	//==============================================================
	// EN: Stack buffer conveyor control
	// PT: Controle das esteiras buffer de pilhas
	//==============================================================
	stackBufferControlState                 : INT;
	stackBufferTargetConveyor               : INT;
	elevatorStackExitClearSensorOld         : BOOL;
	rElevatorStackExitClear                 : BOOL;
	tonStackBufferStopDelay                 : TON;
	tonStackBufferTransferTimeout           : TON;
	tonStackBufferFullSpeedReduction        : TON;
	stackBufferTransferTimeoutPulse         : BOOL;
	
	instTONPaperPressOff: TON;
	instTONPaperPressOn: TON;
	paperPressOnPhase: BOOL;

	// EN: Delays exhaust fan shutdown after line speed drops.
	// PT: Atrasa o desligamento do exaustor após a queda da velocidade da linha.
	instTONSheetConveyor1ExhaustFanStopDelay : TON;
END_VAR

_SystemControl();

_SheetConveyorGroupControl();
_ConveyorSpeedControl();
_SheetConveyor1ExhaustFanControl();

_SheetStackDischargeControl();

_BackstopControl();
_ElevatorControl();
_SheetStackAlignmentBrushControl();
_SheetStackDischargeConveyorControl();
_StackBufferConveyorsControl();
_SheetBrushControl();
_paperPressControl();
_MachineAuxiliary();
_HmiStatus();
_AlarmControl();

//==============================================================
// COMPLEX STACKER — ALARM CONTROL
// EN: Maps internal faults and status conditions to HMI alarm structure.
//==============================================================
METHOD _AlarmControl

VAR
	alarmCompareResult                         : DINT;
	elevatorHomeReleasePermissivesWithoutBackstop : BOOL;
	elevatorUpBlockedByBackstopCondition       : BOOL;
	elevatorUpPermissivesWithoutBackstop       : BOOL;
	elevatorUpRequestActive                    : BOOL;
	hmiAlarmsNotActive                         : hmiAlarmsComplexStacker_TypeStruct;
END_VAR
//==============================================================
// HMI alarms reset / latch logic
//==============================================================

// EN: Detect an actual upward request before the backstop material sensor
//     is applied to the elevator movement permissive.
// PT: Detecta um pedido real de subida antes de aplicar o sensor de material
//     do backstop ao permissivo de movimento do elevador.
elevatorUpRequestActive :=
    (
        (elevatorControlState = 11) AND
        elevatorHomeLimitReached
    ) OR
    (
        (elevatorControlState = 14) AND
        elevatorHomeDischargeComplete AND
        NOT elevatorInPosition AND
        (elevatorRawSpeedRefMmps > 0.0)
    ) OR
    (
        (elevatorControlState = 20) AND
        elevatorManualCommandRequest AND
        elevatorUpCmd AND
        NOT elevatorDownCmd
    ) OR
    (
        (elevatorControlState = 40) AND
        elevatorTargetOverrideActive AND
        NOT elevatorInPosition AND
        (elevatorRawSpeedRefMmps > 0.0)
    );


elevatorUpPermissivesWithoutBackstop :=
    systemRunEnable AND
    safetyCircuitOk AND
    elevatorDriveOk AND
    NOT elevatorFault AND
    NOT elevatorUpperLimit AND
    NOT elevatorUpperSafetyLimit AND
    (
        NOT elevatorHomed OR
        (elevatorPositionMm < machineConfig.elevatorMaxPositionMm)
    );


elevatorHomeReleasePermissivesWithoutBackstop :=
    systemRunEnable AND
    safetyCircuitOk AND
    elevatorDriveOk AND
    NOT elevatorFault AND
    NOT elevatorUpperLimit AND
    NOT elevatorUpperSafetyLimit;


elevatorUpBlockedByBackstopCondition :=
    backstopMaterialInterlockSensor AND
    (
        (
            (elevatorControlState = 11) AND
            elevatorHomeLimitReached AND
            elevatorHomeReleasePermissivesWithoutBackstop
        ) OR
        (
            (elevatorControlState <> 11) AND
            elevatorUpRequestActive AND
            elevatorUpPermissivesWithoutBackstop
        )
    );


// EN: A short delay avoids latching the alarm because of sensor bounce.
// PT: Um pequeno atraso evita memorizar o alarme devido a repique do sensor.
tonElevatorUpBlockedByBackstopAlarm(
    IN := elevatorUpBlockedByBackstopCondition,
    PT := T#500MS
);

IF resetCmd THEN

    // Reset geral dos alarmes
    hmiAlarms := hmiAlarmsNotActive;

ELSE

    //==============================================================
    // 1) General / system alarms
    //==============================================================
    hmiAlarms.safetyCircuitNotOk :=
        hmiAlarms.safetyCircuitNotOk OR
        NOT safetyCircuitOk;

    hmiAlarms.systemFaultActive :=
        hmiAlarms.systemFaultActive OR
        faultActive OR
        (
            backstopRequiredForAutomaticOperation AND
            backstopFault
        ) OR
        elevatorFault OR
        sheetStackDischargeFault OR
        sheetStackDischargeConveyorFault OR
        NOT stackBufferConveyor1DriveOk OR
        NOT stackBufferConveyor2DriveOk OR
        NOT stackBufferConveyor3DriveOk OR
        stackBufferTransferTimeoutPulse;

    hmiAlarms.systemNotEnabled :=
        hmiAlarms.systemNotEnabled OR
        NOT systemRunEnable;

    // EN: These generic safety feedbacks are used only for diagnostics.
    // PT: Estes retornos genéricos de segurança são usados apenas para diagnóstico.
    hmiAlarms.safetyFeedback1NotOk := hmiAlarms.safetyFeedback1NotOk OR NOT safetyFeedBack1;
    hmiAlarms.safetyFeedback2NotOk := hmiAlarms.safetyFeedback2NotOk OR NOT safetyFeedBack2;
    hmiAlarms.safetyFeedback3NotOk := hmiAlarms.safetyFeedback3NotOk OR NOT safetyFeedBack3;
    hmiAlarms.safetyFeedback4NotOk := hmiAlarms.safetyFeedback4NotOk OR NOT safetyFeedBack4;
    hmiAlarms.safetyFeedback5NotOk := hmiAlarms.safetyFeedback5NotOk OR NOT safetyFeedBack5;
    hmiAlarms.safetyFeedback6NotOk := hmiAlarms.safetyFeedback6NotOk OR NOT safetyFeedBack6;
    hmiAlarms.safetyFeedback7NotOk := hmiAlarms.safetyFeedback7NotOk OR NOT safetyFeedBack7;
    hmiAlarms.safetyFeedback8NotOk := hmiAlarms.safetyFeedback8NotOk OR NOT safetyFeedBack8;


    //==============================================================
    // 2) Sheet conveyor group alarms
    //==============================================================
    hmiAlarms.sheetConveyor1DriveNotOk :=
        hmiAlarms.sheetConveyor1DriveNotOk OR
        NOT sheetConveyor1DriveOk;

    hmiAlarms.sheetConveyor2DriveNotOk :=
        hmiAlarms.sheetConveyor2DriveNotOk OR
        NOT sheetConveyor2DriveOk;

    hmiAlarms.sheetConveyor3DriveNotOk :=
        hmiAlarms.sheetConveyor3DriveNotOk OR
        NOT sheetConveyor3DriveOk;

    hmiAlarms.sheetConveyor4DriveNotOk :=
        hmiAlarms.sheetConveyor4DriveNotOk OR
        NOT sheetConveyor4DriveOk;

    hmiAlarms.sheetConveyorGroupFault :=
        hmiAlarms.sheetConveyorGroupFault OR
        NOT safetyCircuitOk OR
        NOT sheetConveyor1DriveOk OR
        NOT sheetConveyor2DriveOk OR
        NOT sheetConveyor3DriveOk OR
        NOT sheetConveyor4DriveOk;


    //==============================================================
    // 2.1) Stack buffer conveyor alarms
    // EN: Buffer drive faults are alarmed without stopping the main
    //     synchronized conveyor group automatically.
    // PT: Falhas dos drives do buffer geram alarme sem parar automaticamente
    //     o grupo principal de esteiras sincronizadas.
    //==============================================================
    hmiAlarms.stackBufferConveyor1DriveNotOk :=
        hmiAlarms.stackBufferConveyor1DriveNotOk OR
        NOT stackBufferConveyor1DriveOk;

    hmiAlarms.stackBufferConveyor2DriveNotOk :=
        hmiAlarms.stackBufferConveyor2DriveNotOk OR
        NOT stackBufferConveyor2DriveOk;

    hmiAlarms.stackBufferConveyor3DriveNotOk :=
        hmiAlarms.stackBufferConveyor3DriveNotOk OR
        NOT stackBufferConveyor3DriveOk;

    hmiAlarms.stackBufferConveyorGroupFault :=
        hmiAlarms.stackBufferConveyorGroupFault OR
        NOT safetyCircuitOk OR
        NOT stackBufferConveyor1DriveOk OR
        NOT stackBufferConveyor2DriveOk OR
        NOT stackBufferConveyor3DriveOk;

    hmiAlarms.stackBufferTransferTimeout :=
        hmiAlarms.stackBufferTransferTimeout OR
        stackBufferTransferTimeoutPulse;

    hmiAlarms.stackBufferFull :=
        hmiAlarms.stackBufferFull OR
        stackBufferFull;

    hmiAlarms.stackBufferSpeedReductionActive :=
        hmiAlarms.stackBufferSpeedReductionActive OR
        lineSpeedReductionRequest;

 //   hmiAlarms.synchronizedConveyorsNotRunning :=
 //       hmiAlarms.synchronizedConveyorsNotRunning OR
 //       (
 //           systemRunEnable AND
 //           NOT synchronizedConveyorsRunning
 //       );


    //==============================================================
    // 3) Sheet stack separation alarms / indications
    //==============================================================
    // Mantido comentado conforme lógica original.
    // Se quiser ativar como latch, use o mesmo padrão:
    //
    // hmiAlarms.sheetStackSeparationNotReady :=
    //     hmiAlarms.sheetStackSeparationNotReady OR
    //     (
    //         systemRunEnable AND
    //         synchronizedConveyorsRunning AND
    //         NOT sheetStackSeparationReady
    //     );
    //
    // hmiAlarms.sheetStackSeparationActive :=
    //     hmiAlarms.sheetStackSeparationActive OR
    //     sheetStackSeparationActive;
    //
    // hmiAlarms.sheetStackBrakeActive :=
    //     hmiAlarms.sheetStackBrakeActive OR
    //     sheetStackBrakeActive;


    //==============================================================
    // 4) Sheet stack discharge sequence alarms / indications
    //==============================================================
    hmiAlarms.sheetStackDischargeFault :=
        hmiAlarms.sheetStackDischargeFault OR
        sheetStackDischargeFault;

    hmiAlarms.sheetStackDischargeLastCycleNotOk :=
        hmiAlarms.sheetStackDischargeLastCycleNotOk OR
        (
            NOT sheetStackDischargeLastCycleOk AND
            sheetStackDischargeLastResultCode <> 0
        );

    hmiAlarms.sheetStackDischargeTimeout :=
        hmiAlarms.sheetStackDischargeTimeout OR
        (
            sheetStackDischargeFault AND
            (sheetStackDischargeLastResultCode = 3)
        );

    hmiAlarms.sheetStackDischargeManualSkip :=
        hmiAlarms.sheetStackDischargeManualSkip OR
        sheetStackDischargeLastResultCode = 2;

    hmiAlarms.sheetStackDischargeWaitSeparationTimeout :=
        hmiAlarms.sheetStackDischargeWaitSeparationTimeout OR
        (
            sheetStackDischargeFault AND
            (sheetStackDischargeLastFaultCode = 10)
        );

    hmiAlarms.sheetStackDischargePositioningTimeout :=
        hmiAlarms.sheetStackDischargePositioningTimeout OR
        (
            sheetStackDischargeFault AND
            (sheetStackDischargeLastFaultCode = 20)
        );

    hmiAlarms.sheetStackDischargeConveyorStartTimeout :=
        hmiAlarms.sheetStackDischargeConveyorStartTimeout OR
        (
            sheetStackDischargeFault AND
            (sheetStackDischargeLastFaultCode = 30)
        );

    hmiAlarms.sheetStackDischargePlatformClearTimeout :=
        hmiAlarms.sheetStackDischargePlatformClearTimeout OR
        (
            sheetStackDischargeFault AND
            (sheetStackDischargeLastFaultCode = 31)
        );

    hmiAlarms.sheetStackDischargeReturnTimeout :=
        hmiAlarms.sheetStackDischargeReturnTimeout OR
        (
            sheetStackDischargeFault AND
            (sheetStackDischargeLastFaultCode = 50)
        );


    //==============================================================
    // 5) Sheet stack discharge conveyor alarms
    //==============================================================
    hmiAlarms.sheetStackDischargeConveyorDriveNotOk :=
        hmiAlarms.sheetStackDischargeConveyorDriveNotOk OR
        NOT sheetStackDischargeConveyorDriveOk;

    hmiAlarms.sheetStackDischargeConveyorFault :=
        hmiAlarms.sheetStackDischargeConveyorFault OR
        sheetStackDischargeConveyorFault;


    //==============================================================
    // 6) Backstop alarms / indications
    //==============================================================
    hmiAlarms.backstopDriveNotOk :=
        hmiAlarms.backstopDriveNotOk OR
        NOT backstopDriveOk;

    hmiAlarms.backstopFault :=
        hmiAlarms.backstopFault OR
        backstopFault;

    hmiAlarms.backstopNotHomed :=
        hmiAlarms.backstopNotHomed OR
        (
            systemRunEnable AND
            backstopAutoCmd AND
            NOT backstopHomed AND
            NOT backstopAutoHomePending AND
            NOT (
                (backstopControlState >= 10) AND
                (backstopControlState <= 14)
            )
        );

    hmiAlarms.backstopHomingTimeout :=
        hmiAlarms.backstopHomingTimeout OR
        (
            backstopFault AND
            (backstopFaultCode = 3)
        );

    hmiAlarms.backstopInvalidHomeDirection :=
        hmiAlarms.backstopInvalidHomeDirection OR
        (
            backstopFault AND
            (backstopFaultCode = 5)
        );

    (*
    hmiAlarms.backstopNotInPosition :=
        hmiAlarms.backstopNotInPosition OR
        (
            systemRunEnable AND
            backstopAutoCmd AND
            backstopHomed AND
            NOT backstopInPosition AND
            NOT backstopTargetOverrideActive
        );
    *)

    hmiAlarms.backstopSafeMaxLimitActive :=
        hmiAlarms.backstopSafeMaxLimitActive OR
        backstopSafeMaxLimit;

    hmiAlarms.backstopSafeMinLimitActive :=
        hmiAlarms.backstopSafeMinLimitActive OR
        backstopSafeMinLimit;

    (*
    hmiAlarms.backstopMaxLimitActive :=
        hmiAlarms.backstopMaxLimitActive OR
        backstopMaxLimit;

    hmiAlarms.backstopMinLimitActive :=
        hmiAlarms.backstopMinLimitActive OR
        backstopMinLimit;

    hmiAlarms.backstopManualInterventionActive :=
        hmiAlarms.backstopManualInterventionActive OR
        backstopManualInterventionActive;
    *)


    //==============================================================
    // 7) Elevator alarms / indications
    //==============================================================
    hmiAlarms.elevatorDriveNotOk :=
        hmiAlarms.elevatorDriveNotOk OR
        NOT elevatorDriveOk;

    hmiAlarms.elevatorFault :=
        hmiAlarms.elevatorFault OR
        elevatorFault;

    hmiAlarms.elevatorNotHomed :=
        hmiAlarms.elevatorNotHomed OR
        (
            systemRunEnable AND
            elevatorAutoCmd AND
            NOT elevatorHomed AND
            NOT elevatorAutoHomePending AND
            NOT (
                (elevatorControlState >= 10) AND
                (elevatorControlState <= 14)
            )
        );

    hmiAlarms.elevatorHomingTimeout :=
        hmiAlarms.elevatorHomingTimeout OR
        (
            elevatorFault AND
            (elevatorFaultCode = 3)
        );

    hmiAlarms.elevatorUpBlockedByBackstopMaterialInterlock :=
        hmiAlarms.elevatorUpBlockedByBackstopMaterialInterlock OR
        tonElevatorUpBlockedByBackstopAlarm.Q;

//    hmiAlarms.elevatorNotInPosition :=
//        hmiAlarms.elevatorNotInPosition OR
//        (
//            systemRunEnable AND
//            elevatorAutoCmd AND
//            elevatorHomed AND
//            NOT elevatorInPosition
//        );

    hmiAlarms.elevatorUpperSafetyLimitActive :=
        hmiAlarms.elevatorUpperSafetyLimitActive OR
        elevatorUpperSafetyLimit;

    hmiAlarms.elevatorLowerSafetyLimitActive :=
        hmiAlarms.elevatorLowerSafetyLimitActive OR
        elevatorLowerSafetyLimit;

    (*
    hmiAlarms.elevatorUpperLimitActive :=
        hmiAlarms.elevatorUpperLimitActive OR
        elevatorUpperLimit;

    hmiAlarms.elevatorLowerLimitActive :=
        hmiAlarms.elevatorLowerLimitActive OR
        elevatorLowerLimit;
    *)

END_IF;


// EN: The general output follows every latched field in the alarm structure.
// PT: A saída geral acompanha qualquer campo memorizado na estrutura de alarmes.
alarmCompareResult := MEMCMP(
    pBuf1 := ADR(hmiAlarmsNotActive),
    pBuf2 := ADR(hmiAlarms),
    n := SIZEOF(hmiAlarms)
);

alarmActive := alarmCompareResult <> 0;
END_METHOD

//==============================================================
// COMPLEX STACKER — BACKSTOP CONTROL
// EN: Controls the backstop axis with homing, manual movement,
//     automatic positioning, override positioning and protections.
//
// Signed speed convention:
// Positive = open
// Negative = close
//
// State code:
// 0  = STOP
// 10 = HOME_FAST_SEARCH
// 11 = HOME_SLOW_EXIT_SENSOR
// 12 = HOME_SET_ENCODER
// 13 = HOME_WAIT_AFTER_SET
// 14 = HOME_MOVE_TO_TARGET
// 20 = MANUAL
// 30 = AUTO_POSITION
// 40 = FAULT
//==============================================================
METHOD _BackstopControl



//==============================================================
// 1) Default internal commands
//==============================================================
// EN: Internal signed speed is reset every scan and set by the active state.
//     Positive = open, negative = close.
backstopSignedSpeedRefMmps := 0.0;

// EN: Internal trigger for encoder set pulse.
backstopSetEncoderPositionTrigger := FALSE;


//==============================================================
// 2) Edge detection
//==============================================================
// EN: Home can be requested manually by HMI or automatically by _SystemControl.
//     Automatic home is accepted only when backstopAutoCmd is enabled.
//     Movement is allowed only when master system run is enabled.
backstopHomeRequestCombined :=
    systemRunEnable AND
    (
        backstopHomeCmd OR
        (
            backstopAutoCmd AND
            backstopAutoHomeRequest
        )
    );

// EN: The automatic pulse is accepted directly so a maintained manual home
//     command cannot hide the mandatory start-triggered request.
// PT: O pulso automático é aceito diretamente para que um comando manual de
//     home mantido não esconda o pedido obrigatório gerado pela partida.
rBackstopHome :=
    (
        backstopHomeRequestCombined AND
        NOT backstopHomeRequestCombinedOld
    ) OR
    (
        systemRunEnable AND
        backstopAutoCmd AND
        backstopAutoHomeRequest
    );

backstopHomeRequestCombinedOld :=
    backstopHomeRequestCombined;


// EN: Execute positioning command edge.
//     This command only generates movement when system is enabled and backstop auto is enabled.
rBackstopExecutePositioning :=
    systemRunEnable AND
    backstopExecutePositioningCmd AND
    NOT backstopExecutePositioningCmdOld;

backstopExecutePositioningCmdOld := backstopExecutePositioningCmd;


// EN: Override falling edge.
//     Used as fallback to return to programmed position if override is released.
backstopTargetOverrideFallingEdge :=
    backstopTargetOverrideOld AND NOT backstopTargetOverrideActive;

backstopTargetOverrideOld := backstopTargetOverrideActive;


//==============================================================
// 3) Home limit selection and edge detection
//==============================================================
// EN: Home limit depends on configured homing direction.
IF machineConfig.backstopHomeDirection > 0 THEN

    backstopHomeLimitReached := backstopMaxLimit;

ELSIF machineConfig.backstopHomeDirection < 0 THEN

    backstopHomeLimitReached := backstopMinLimit;

ELSE

    backstopHomeLimitReached := FALSE;

END_IF;


// EN: Falling edge is used after the home limit has been reached.
backstopHomeLimitFallingEdge :=
    backstopHomeLimitOld AND NOT backstopHomeLimitReached;

backstopHomeLimitOld := backstopHomeLimitReached;


//==============================================================
// 4) Movement permissions
//==============================================================
backstopOpenAllowed :=
    systemRunEnable AND
    safetyCircuitOk AND
    backstopDriveOk AND
    NOT backstopMaxLimit AND
    NOT backstopSafeMaxLimit AND
    (
        (NOT backstopHomed) OR
        (backstopPositionMm < machineConfig.backstopMaxPositionMm)
    );

backstopCloseAllowed :=
    systemRunEnable AND
    safetyCircuitOk AND
    backstopDriveOk AND
    NOT backstopMinLimit AND
    NOT backstopSafeMinLimit AND
    (
        (NOT backstopHomed) OR
        (backstopPositionMm > machineConfig.backstopMinPositionMm)
    );


// EN: During homing, the normal home limit is allowed.
//     Only the safe limit blocks movement.
IF machineConfig.backstopHomeDirection > 0 THEN

    backstopHomeMoveAllowed :=
        systemRunEnable AND
        safetyCircuitOk AND
        backstopDriveOk AND
        NOT backstopSafeMaxLimit;

ELSIF machineConfig.backstopHomeDirection < 0 THEN

    backstopHomeMoveAllowed :=
        systemRunEnable AND
        safetyCircuitOk AND
        backstopDriveOk AND
        NOT backstopSafeMinLimit;

ELSE

    backstopHomeMoveAllowed := FALSE;

END_IF;


//==============================================================
// 5) Programmed / override target calculation
//==============================================================
// EN: Programmed target follows sheet length plus mechanical offset.
//     This value can change, but it does not move the backstop by itself.
backstopProgrammedTargetPositionMm :=
    LIMIT(
        machineConfig.backstopMinPositionMm,
        MAX(0.0, sheetLengthMm) + machineConfig.backstopSheetLengthOffsetMm,
        machineConfig.backstopMaxPositionMm
    );


// EN: Before homing, keep the latched target updated with programmed target.
//     This avoids an invalid old target after power-up.
IF NOT backstopHomed THEN

    backstopLatchedTargetPositionMm := backstopProgrammedTargetPositionMm;

END_IF;


//==============================================================
// 5.1) Automatic positioning request handling
//==============================================================
// EN: Auto mode only enables positioning. It does not execute positioning.
//     Normal positioning must be requested by backstopExecutePositioningCmd.
//     Override positioning is requested by the automatic cycle.
IF NOT systemRunEnable THEN

    backstopPositioningRequestActive := FALSE;


ELSIF NOT backstopAutoCmd THEN

    backstopPositioningRequestActive := FALSE;


ELSIF backstopTargetOverrideActive THEN

    // EN: Override has priority. Clear normal positioning request.
    backstopPositioningRequestActive := FALSE;


ELSIF rBackstopExecutePositioning THEN

    // EN: Latch current programmed target only when execute command is received.
    backstopLatchedTargetPositionMm := backstopProgrammedTargetPositionMm;
    backstopPositioningRequestActive := TRUE;


ELSIF backstopTargetOverrideFallingEdge THEN

    // EN: Fallback after override release.
    //     The discharge sequence should normally keep override active
    //     during return. If override is released unexpectedly, return to
    //     programmed position automatically.
    backstopLatchedTargetPositionMm := backstopProgrammedTargetPositionMm;
    backstopPositioningRequestActive := TRUE;

END_IF;


//==============================================================
// 5.2) Active target selection
//==============================================================
// EN: Discharge override is accepted only while the backstop is in automatic.
//     In manual mode the backstop is completely independent from the cycle.
// PT: O override de descarte é aceito somente com o backstop em automático.
//     No modo manual o backstop fica completamente independente do ciclo.
IF systemRunEnable AND
   backstopAutoCmd AND
   backstopTargetOverrideActive THEN

    backstopTargetPositionMm :=
        LIMIT(
            machineConfig.backstopMinPositionMm,
            backstopTargetOverridePositionMm,
            machineConfig.backstopMaxPositionMm
        );

ELSE

    backstopTargetPositionMm :=
        LIMIT(
            machineConfig.backstopMinPositionMm,
            backstopLatchedTargetPositionMm,
            machineConfig.backstopMaxPositionMm
        );

END_IF;


//==============================================================
// 5.4) Home running flag
//==============================================================
IF (backstopControlState = 10) OR
   (backstopControlState = 11) OR
   (backstopControlState = 12) OR
   (backstopControlState = 13) OR
   (backstopControlState = 14) THEN

    backstopHomeRunning := TRUE;

ELSE

    backstopHomeRunning := FALSE;

END_IF;


//==============================================================
// 6) Position error calculation
//==============================================================
backstopPositionErrorMm :=
    backstopTargetPositionMm - backstopPositionMm;

backstopAbsPositionErrorMm :=
    ABS(backstopPositionErrorMm);

backstopInPosition :=
    backstopHomed AND
    (backstopAbsPositionErrorMm <= machineConfig.backstopPositionToleranceMm);


//==============================================================
// 7) Reset fault command
//==============================================================
IF resetCmd THEN

    IF safetyCircuitOk AND
       backstopDriveOk AND
       NOT backstopSafeMaxLimit AND
       NOT backstopSafeMinLimit THEN

        backstopFault := FALSE;
        backstopFaultCode := 0;

        IF backstopControlState = 40 THEN
            backstopControlState := 0;
        END_IF

    END_IF

END_IF;


//==============================================================
// 8) General protection
//==============================================================
IF NOT safetyCircuitOk THEN

    backstopState := 'SAFETY_OFF';

    tonBackstopHomingTimeout(IN := FALSE);
    tonBackstopHomeSettleDelay(IN := FALSE);

    backstopFault := TRUE;
    backstopFaultCode := 2;
    backstopControlState := 40;


ELSIF NOT backstopDriveOk THEN

    backstopState := 'DRIVE_NOT_OK';

    tonBackstopHomingTimeout(IN := FALSE);
    tonBackstopHomeSettleDelay(IN := FALSE);

    backstopFault := TRUE;
    backstopFaultCode := 1;
    backstopControlState := 40;


ELSIF backstopSafeMaxLimit THEN

    backstopState := 'SAFE_MAX_LIMIT';

    tonBackstopHomingTimeout(IN := FALSE);
    tonBackstopHomeSettleDelay(IN := FALSE);

    backstopFault := TRUE;
    backstopFaultCode := 6;
    backstopControlState := 40;


ELSIF backstopSafeMinLimit THEN

    backstopState := 'SAFE_MIN_LIMIT';

    tonBackstopHomingTimeout(IN := FALSE);
    tonBackstopHomeSettleDelay(IN := FALSE);

    backstopFault := TRUE;
    backstopFaultCode := 7;
    backstopControlState := 40;


ELSIF machineConfig.backstopHomeDirection = 0 THEN

    backstopState := 'INVALID_HOME_DIR';

    tonBackstopHomingTimeout(IN := FALSE);
    tonBackstopHomeSettleDelay(IN := FALSE);

    backstopFault := TRUE;
    backstopFaultCode := 5;
    backstopControlState := 40;


ELSIF NOT systemRunEnable THEN

    // EN: Master stop disables movement without generating an axis fault.
    backstopState := 'SYSTEM_DISABLED';

    backstopSignedSpeedRefMmps := 0.0;

    tonBackstopHomingTimeout(IN := FALSE);
    tonBackstopHomeSettleDelay(IN := FALSE);

    backstopPositioningRequestActive := FALSE;

    IF backstopControlState <> 40 THEN
        backstopControlState := 0;
    END_IF


ELSE

    //==============================================================
    // 9) Mode selection
    //==============================================================
    // EN: Homing has priority over manual and automatic positioning.
    IF rBackstopHome AND NOT backstopFault THEN
        backstopControlState := 10;

        // EN: Consume the pending request only after homing is accepted.
        // PT: Consome o pedido pendente somente após o homing ser aceito.
        backstopAutoHomePending := FALSE;
    END_IF;


    //==============================================================
    // 10) Backstop state machine
    //==============================================================
    CASE backstopControlState OF

        0: // STOP
            backstopState := 'STOP';

            tonBackstopHomingTimeout(IN := FALSE);
            tonBackstopHomeSettleDelay(IN := FALSE);

            // EN: Manual is allowed even with auto enabled,
            //     but not during an automatic cycle override.
            IF (backstopOpenCmd OR backstopCloseCmd) AND
               NOT (
                   backstopAutoCmd AND
                   backstopTargetOverrideActive
               ) THEN

                backstopControlState := 20;


            ELSIF backstopAutoCmd AND
                  (
                      backstopTargetOverrideActive OR
                      backstopPositioningRequestActive
                  ) THEN

                backstopControlState := 30;

            END_IF


        10: // HOME_FAST_SEARCH
            backstopState := 'HOME_FAST';

            backstopHomed := FALSE;
            backstopInPosition := FALSE;

            tonBackstopHomeSettleDelay(IN := FALSE);

            tonBackstopHomingTimeout(
                IN := TRUE,
                PT := machineConfig.backstopHomingTimeout
            );

            IF tonBackstopHomingTimeout.Q THEN

                backstopSignedSpeedRefMmps := 0.0;

                tonBackstopHomingTimeout(IN := FALSE);

                backstopFault := TRUE;
                backstopFaultCode := 3;

                backstopState := 'HOME_TIMEOUT';
                backstopControlState := 40;


            ELSIF backstopHomeLimitReached THEN

                backstopSignedSpeedRefMmps := 0.0;

                backstopControlState := 11;


            ELSE

                IF backstopHomeMoveAllowed THEN

                    IF machineConfig.backstopHomeDirection > 0 THEN

                        backstopSignedSpeedRefMmps :=
                            ABS(machineConfig.backstopHomingSpeedMmps);

                    ELSE

                        backstopSignedSpeedRefMmps :=
                            -ABS(machineConfig.backstopHomingSpeedMmps);

                    END_IF

                ELSE

                    backstopSignedSpeedRefMmps := 0.0;

                END_IF

            END_IF


        11: // HOME_SLOW_EXIT_SENSOR
            backstopState := 'HOME_SLOW_EXIT';

            tonBackstopHomeSettleDelay(IN := FALSE);

            tonBackstopHomingTimeout(
                IN := TRUE,
                PT := machineConfig.backstopHomingTimeout
            );

            IF tonBackstopHomingTimeout.Q THEN

                backstopSignedSpeedRefMmps := 0.0;

                tonBackstopHomingTimeout(IN := FALSE);

                backstopFault := TRUE;
                backstopFaultCode := 3;

                backstopState := 'HOME_TIMEOUT';
                backstopControlState := 40;


            ELSIF backstopHomeLimitFallingEdge THEN

                backstopSignedSpeedRefMmps := 0.0;

                tonBackstopHomingTimeout(IN := FALSE);

                backstopControlState := 12;


            ELSE

                IF backstopHomeMoveAllowed THEN

                    IF machineConfig.backstopHomeDirection > 0 THEN

                        backstopSignedSpeedRefMmps :=
                            -ABS(machineConfig.backstopMinMoveSpeedMmps);

                    ELSE

                        backstopSignedSpeedRefMmps :=
                            ABS(machineConfig.backstopMinMoveSpeedMmps);

                    END_IF

                ELSE

                    backstopSignedSpeedRefMmps := 0.0;

                END_IF

            END_IF


        12: // HOME_SET_ENCODER
            backstopState := 'HOME_SET_ENCODER';

            backstopSignedSpeedRefMmps := 0.0;

            tonBackstopHomingTimeout(IN := FALSE);
            tonBackstopHomeSettleDelay(IN := FALSE);

            // EN: Set encoder to configured known home position.
            backstopSetEncoderPositionTrigger := TRUE;
            backstopSetEncoderPositionMm := machineConfig.backstopHomePositionMm;

            backstopHomed := TRUE;
            backstopFault := FALSE;
            backstopFaultCode := 0;

            // EN: After homing, latch current programmed target for home move.
            backstopLatchedTargetPositionMm := backstopProgrammedTargetPositionMm;
            backstopPositioningRequestActive := TRUE;

            // EN: Homing cancels previous manual intervention memory.
            backstopManualInterventionActive := FALSE;
            backstopManualInterventionPositionMm := 0.0;

            backstopControlState := 13;


        13: // HOME_WAIT_AFTER_SET
            backstopState := 'HOME_WAIT';

            backstopSignedSpeedRefMmps := 0.0;

            tonBackstopHomingTimeout(IN := FALSE);

            // EN: Fixed wait after encoder set.
            tonBackstopHomeSettleDelay(
                IN := TRUE,
                PT := T#5S
            );

            IF tonBackstopHomeSettleDelay.Q THEN

                tonBackstopHomeSettleDelay(IN := FALSE);

                backstopControlState := 14;

            END_IF


        14: // HOME_MOVE_TO_TARGET
            backstopState := 'HOME_TO_TARGET';

            tonBackstopHomingTimeout(IN := FALSE);
            tonBackstopHomeSettleDelay(IN := FALSE);

            // EN: Move to the latched programmed target after homing.
            IF backstopInPosition THEN

                backstopSignedSpeedRefMmps := 0.0;

                backstopPositioningRequestActive := FALSE;

                // EN: Home positioning completed, no manual intervention pending.
                backstopManualInterventionActive := FALSE;
                backstopManualInterventionPositionMm := 0.0;

                backstopControlState := 0;


            ELSE

                backstopRawSpeedRefMmps :=
                    backstopPositionErrorMm * machineConfig.backstopPositionKp;

                backstopRawSpeedRefMmps :=
                    LIMIT(
                        -ABS(machineConfig.backstopAutoMaxSpeedMmps),
                        backstopRawSpeedRefMmps,
                        ABS(machineConfig.backstopAutoMaxSpeedMmps)
                    );

                IF ABS(backstopRawSpeedRefMmps) <
                   ABS(machineConfig.backstopMinMoveSpeedMmps) THEN

                    IF backstopPositionErrorMm > 0.0 THEN

                        backstopRawSpeedRefMmps :=
                            ABS(machineConfig.backstopMinMoveSpeedMmps);

                    ELSE

                        backstopRawSpeedRefMmps :=
                            -ABS(machineConfig.backstopMinMoveSpeedMmps);

                    END_IF

                END_IF

                IF (backstopRawSpeedRefMmps > 0.0) AND backstopOpenAllowed THEN

                    backstopSignedSpeedRefMmps := backstopRawSpeedRefMmps;

                ELSIF (backstopRawSpeedRefMmps < 0.0) AND backstopCloseAllowed THEN

                    backstopSignedSpeedRefMmps := backstopRawSpeedRefMmps;

                ELSE

                    backstopSignedSpeedRefMmps := 0.0;

                END_IF

            END_IF


        20: // MANUAL
            backstopState := 'MANUAL';

            tonBackstopHomingTimeout(IN := FALSE);
            tonBackstopHomeSettleDelay(IN := FALSE);

            // EN: An automatic override cancels manual control only when
            //     the backstop itself is enabled in automatic mode.
            // PT: O override automático cancela o controle manual somente
            //     quando o próprio backstop está habilitado em automático.
            IF backstopAutoCmd AND
               backstopTargetOverrideActive THEN

                backstopSignedSpeedRefMmps := 0.0;
                backstopControlState := 30;


            ELSIF backstopOpenCmd AND backstopCloseCmd THEN

                backstopSignedSpeedRefMmps := 0.0;


            ELSIF backstopOpenCmd THEN

                IF backstopOpenAllowed THEN

                    backstopSignedSpeedRefMmps :=
                        ABS(machineConfig.backstopManualSpeedMmps);

                    // EN: Store last manual intervention position.
                    //     This is updated while the operator holds the manual command.
                    backstopManualInterventionActive := TRUE;
                    backstopManualInterventionPositionMm := backstopPositionMm;

                ELSE

                    backstopSignedSpeedRefMmps := 0.0;

                END_IF


            ELSIF backstopCloseCmd THEN

                IF backstopCloseAllowed THEN

                    backstopSignedSpeedRefMmps :=
                        -ABS(machineConfig.backstopManualSpeedMmps);

                    // EN: Store the last manual intervention position.
                    //     The discharge opening uses the greater value between the
                    //     current mechanical position and this stored position.
                    // PT: Memoriza a última posição de intervenção manual.
                    //     A abertura de descarga usa o maior valor entre a posição
                    //     mecânica atual e esta posição memorizada.
                    backstopManualInterventionActive := TRUE;
                    backstopManualInterventionPositionMm := backstopPositionMm;

                ELSE

                    backstopSignedSpeedRefMmps := 0.0;

                END_IF


            ELSE

                backstopSignedSpeedRefMmps := 0.0;

                // EN: After manual command release, do not automatically return
                //     to programmed position. Wait for execute positioning command.
                backstopPositioningRequestActive := FALSE;

                backstopControlState := 0;

            END_IF


        30: // AUTO_POSITION
            backstopState := 'AUTO_POSITION';

            tonBackstopHomingTimeout(IN := FALSE);
            tonBackstopHomeSettleDelay(IN := FALSE);

            // EN: Manual mode always cancels automatic positioning,
            //     regardless of any external override request.
            // PT: O modo manual sempre cancela o posicionamento automático,
            //     independentemente de qualquer pedido externo de override.
            IF NOT backstopAutoCmd THEN

                backstopSignedSpeedRefMmps := 0.0;
                backstopPositioningRequestActive := FALSE;
                backstopControlState := 0;


            ELSIF NOT backstopHomed THEN

                backstopSignedSpeedRefMmps := 0.0;
                backstopState := 'AUTO_NO_HOME';


            ELSIF (backstopOpenCmd OR backstopCloseCmd) AND
                  NOT backstopTargetOverrideActive THEN

                // EN: Manual has priority only outside automatic cycle override.
                backstopSignedSpeedRefMmps := 0.0;
                backstopPositioningRequestActive := FALSE;
                backstopControlState := 20;


            ELSIF NOT backstopTargetOverrideActive AND
                  NOT backstopPositioningRequestActive THEN

                // EN: Auto enabled but no positioning command active.
                backstopSignedSpeedRefMmps := 0.0;
                backstopControlState := 0;


            ELSIF backstopInPosition THEN

                backstopSignedSpeedRefMmps := 0.0;

                // EN: Normal positioning command ends when target is reached.
                //     Override remains controlled by the automatic cycle.
                IF NOT backstopTargetOverrideActive THEN

                    backstopPositioningRequestActive := FALSE;

                    // EN: If the backstop returned to programmed target,
                    //     clear previous manual intervention memory.
                    backstopManualInterventionActive := FALSE;
                    backstopManualInterventionPositionMm := 0.0;

                    backstopControlState := 0;

                END_IF


            ELSE

                backstopRawSpeedRefMmps :=
                    backstopPositionErrorMm * machineConfig.backstopPositionKp;

                backstopRawSpeedRefMmps :=
                    LIMIT(
                        -ABS(machineConfig.backstopAutoMaxSpeedMmps),
                        backstopRawSpeedRefMmps,
                        ABS(machineConfig.backstopAutoMaxSpeedMmps)
                    );

                IF ABS(backstopRawSpeedRefMmps) <
                   ABS(machineConfig.backstopMinMoveSpeedMmps) THEN

                    IF backstopPositionErrorMm > 0.0 THEN

                        backstopRawSpeedRefMmps :=
                            ABS(machineConfig.backstopMinMoveSpeedMmps);

                    ELSE

                        backstopRawSpeedRefMmps :=
                            -ABS(machineConfig.backstopMinMoveSpeedMmps);

                    END_IF

                END_IF

                IF (backstopRawSpeedRefMmps > 0.0) AND backstopOpenAllowed THEN

                    backstopSignedSpeedRefMmps := backstopRawSpeedRefMmps;

                ELSIF (backstopRawSpeedRefMmps < 0.0) AND backstopCloseAllowed THEN

                    backstopSignedSpeedRefMmps := backstopRawSpeedRefMmps;

                ELSE

                    backstopSignedSpeedRefMmps := 0.0;

                END_IF

            END_IF


        40: // FAULT
            backstopState := 'FAULT';

            backstopSignedSpeedRefMmps := 0.0;

            tonBackstopHomingTimeout(IN := FALSE);
            tonBackstopHomeSettleDelay(IN := FALSE);

            backstopPositioningRequestActive := FALSE;

            IF resetCmd AND
               safetyCircuitOk AND
               backstopDriveOk AND
               NOT backstopSafeMaxLimit AND
               NOT backstopSafeMinLimit THEN

                backstopFault := FALSE;
                backstopFaultCode := 0;
                backstopControlState := 0;

            END_IF


    ELSE

        backstopControlState := 0;

    END_CASE;

END_IF;


//==============================================================
// 11) Encoder set pulse
//==============================================================
// EN: Extend encoder set command to ensure the encoder block sees it.
tpBackstopSetEncoderPosition(
    IN := backstopSetEncoderPositionTrigger,
    PT := machineConfig.backstopSetEncoderPulseTime
);

backstopSetEncoderPosition := tpBackstopSetEncoderPosition.Q;


//==============================================================
// 12) Backstop drive direction and speed outputs
//==============================================================
// EN: Convert signed internal speed command into direction outputs
//     and positive speed reference.
IF systemRunEnable AND
   safetyCircuitOk AND
   backstopDriveOk AND
   NOT backstopFault AND
   (ABS(backstopSignedSpeedRefMmps) >= machineConfig.backstopRunMinSpeedMmps) THEN

    // EN: The servo receives the signed speed reference directly.
    // PT: O servo recebe diretamente a referência de velocidade com sinal.
    backstopSpeedRefMmps := backstopSignedSpeedRefMmps;

    backstopRunFw :=
        backstopSignedSpeedRefMmps > 0.0;

    backstopRunRev :=
        backstopSignedSpeedRefMmps < 0.0;

ELSE

    backstopSpeedRefMmps := 0.0;

    backstopRunFw := FALSE;
    backstopRunRev := FALSE;

END_IF;

// EN: Enable the servo with the stacker system; drive-ready feedback is not used here
//     because it would create a circular enable dependency.
// PT: Habilita o servo com o sistema do stacker; o retorno de drive pronto não é usado
//     aqui porque criaria uma dependência circular de habilitação.
backstopDriveEnable := systemRunEnable AND safetyCircuitOk;


//==============================================================
// 13) Backstop plate lift solenoid
//==============================================================
// EN: Lift the backstop plate during backstop movement and homing.
//     Discharge conveyor protection can be ORed after all methods are called.
IF systemRunEnable AND
   (
       backstopRunFw OR
       backstopRunRev OR
       sheetStackDischargeActive OR
       (backstopControlState = 10) OR
       (backstopControlState = 11) OR
       (backstopControlState = 12) OR
       (backstopControlState = 13) OR
       (backstopControlState = 14)
   ) THEN

    backstopPlateUpSolenoid := TRUE;
    instTONBackstopDownDelay.IN := FALSE;

ELSE

    instTONBackstopDownDelay.IN := TRUE;

    IF instTONBackstopDownDelay.Q THEN
        backstopPlateUpSolenoid := FALSE;
    END_IF

END_IF;

instTONBackstopDownDelay(PT := T#200MS);
END_METHOD

//==============================================================
// COMPLEX STACKER — SPEED REFERENCE GENERATOR
// EN: Generates synchronized and sheet-stack separation speed references [m/min].
//==============================================================
METHOD _ConveyorSpeedControl
VAR
    packageGapReady                   : BOOL;
    validCycleTimeS                   : REAL;

    sheetConveyorsSpeedUpReferenceMPM : REAL;

    sheetConveyor1BaseSpeedMPM        : REAL;
    sheetConveyor2BaseSpeedMPM        : REAL;
    sheetConveyor3BaseSpeedMPM        : REAL;
    sheetConveyor4BaseSpeedMPM        : REAL;
END_VAR


//==============================================================
// 1) Default event pulses
//==============================================================
sheetStackSeparationStarted         := FALSE;
sheetStackSeparationFinished        := FALSE;

sheetConveyor2SeparationStarted     := FALSE;
sheetConveyor2SeparationFinished    := FALSE;

sheetConveyor3SeparationStarted     := FALSE;
sheetConveyor3SeparationFinished    := FALSE;

sheetConveyor4SeparationStarted     := FALSE;
sheetConveyor4SeparationFinished    := FALSE;


//==============================================================
// 2) Accepted unload event
//==============================================================
// EN: The separation state machine is started only by
//     dischargeRequestAccepted, generated by the discharge controller.
// PT: A máquina de estados de separação é iniciada somente por
//     dischargeRequestAccepted, gerado pelo controle de descarga.


//==============================================================
// 3) Enable and scan time
//==============================================================
speedControlEnabled :=
    sheetConveyor1Run AND
    sheetConveyor2Run AND
    sheetConveyor3Run AND
    sheetConveyor4Run AND
    safetyCircuitOk;

rampReset := NOT speedControlEnabled;


// EN: Read PLC scan time using OSCAT CYCLE_TIME.
instCycleTime(
    RST := resetCmd
);


// EN: Convert last cycle time from TIME/ms to seconds.
scanTimeMs := TIME_TO_REAL(instCycleTime.ct_last);

validCycleTimeS :=
    LIMIT(
        0.001,
        scanTimeMs / 1000.0,
        20.0
    );

scanTimeS := validCycleTimeS;


//==============================================================
// 4) Sheet length conversion
//==============================================================
// EN: Sheet length is kept converted for other calculations,
//     but it is no longer used as the separation tracking target.
sheetLengthM := MAX(0.0, sheetLengthMm) / 1000.0;


//==============================================================
// 5) Select effective line speed during package discharge
//==============================================================
effectiveLineSpeedMPM := MAX(0.0, lineSpeedMPM);

// EN: While package separation is active, a low line speed is replaced by
//     the configured threshold. Outside separation, the actual line speed is used.
// PT: Durante a separação da pilha, uma velocidade baixa da linha é substituída
//     pelo limite configurado. Fora da separação, usa-se a velocidade real da linha.
IF packageSeparationState <> 0 THEN

    effectiveLineSpeedMPM :=
        MAX(
            effectiveLineSpeedMPM,
            MAX(0.0, machineConfig.packageDischargeLineSpeedThresholdMPM)
        );

END_IF;


//==============================================================
// 6) Calculate normal stacker speed
//==============================================================
IF speedControlEnabled THEN

    normalStackerSpeedMPM :=
        LIMIT(
            machineConfig.minimumSpeedMPM,
            effectiveLineSpeedMPM *
                MAX(0.0, machineConfig.stackerSpeedRatio),
            machineConfig.maximumSpeedMPM
        );

ELSE

    normalStackerSpeedMPM := 0.0;

END_IF;


//==============================================================
// 7) Calculate normal speed for each conveyor
//==============================================================
sheetConveyor1NormalSpeedMPM :=
    normalStackerSpeedMPM *
    MAX(0.0, machineConfig.sheetConveyor1SpeedTrim);

sheetConveyor2NormalSpeedMPM :=
    normalStackerSpeedMPM *
    MAX(0.0, machineConfig.sheetConveyor2SpeedTrim);

sheetConveyor3NormalSpeedMPM :=
    normalStackerSpeedMPM *
    MAX(0.0, machineConfig.sheetConveyor3SpeedTrim);

sheetConveyor4NormalSpeedMPM :=
    normalStackerSpeedMPM *
    MAX(0.0, machineConfig.sheetConveyor4SpeedTrim);


//==============================================================
// 6.1) Sheet conveyors speed-up reference
//==============================================================
// EN: Speed-up is added directly to conveyors 1/2/3 references.
//     It can work even when line speed is zero, as long as the
//     conveyor group is enabled.
IF speedControlEnabled AND sheetConveyorsSpeedUpCmd THEN

    sheetConveyorsSpeedUpReferenceMPM :=
        MAX(0.0, machineConfig.sheetConveyorsSpeedUpMPM);

ELSE

    sheetConveyorsSpeedUpReferenceMPM := 0.0;

END_IF;


//==============================================================
// 6.2) Base speed references including speed-up
//==============================================================
// EN: Base speed is the synchronized conveyor speed plus operator speed-up.
//     Separation tracking must use this base speed as reference.
sheetConveyor1BaseSpeedMPM :=
    sheetConveyor1NormalSpeedMPM + sheetConveyorsSpeedUpReferenceMPM;

sheetConveyor2BaseSpeedMPM :=
    sheetConveyor2NormalSpeedMPM + sheetConveyorsSpeedUpReferenceMPM;

sheetConveyor3BaseSpeedMPM :=
    sheetConveyor3NormalSpeedMPM + sheetConveyorsSpeedUpReferenceMPM;

sheetConveyor4BaseSpeedMPM :=
    sheetConveyor4NormalSpeedMPM + sheetConveyorsSpeedUpReferenceMPM;


//==============================================================
// 7) Calculate separation high speed
//==============================================================
// EN: Gap speed also receives the same speed-up reference.
//     This preserves the real gap differential while allowing operator boost.
sheetConveyor1GapSpeedMPM :=
    (sheetConveyor1NormalSpeedMPM * MAX(0.0, machineConfig.packageGapSpeedRatio)) +
    machineConfig.packageGapSpeedOffsetMPM +
    sheetConveyorsSpeedUpReferenceMPM;

sheetConveyor2GapSpeedMPM :=
    (sheetConveyor2NormalSpeedMPM * MAX(0.0, machineConfig.packageGapSpeedRatio)) +
    machineConfig.packageGapSpeedOffsetMPM +
    sheetConveyorsSpeedUpReferenceMPM;

sheetConveyor3GapSpeedMPM :=
    (sheetConveyor3NormalSpeedMPM * MAX(0.0, machineConfig.packageGapSpeedRatio)) +
    machineConfig.packageGapSpeedOffsetMPM +
    sheetConveyorsSpeedUpReferenceMPM;

sheetConveyor4GapSpeedMPM :=
    (sheetConveyor4NormalSpeedMPM * MAX(0.0, machineConfig.packageGapSpeedRatio)) +
    machineConfig.packageGapSpeedOffsetMPM +
    sheetConveyorsSpeedUpReferenceMPM;


//==============================================================
// 8) Calculate separation tracking target distances
//==============================================================
// EN: Separation tracking target is based on each conveyor length.
sheetConveyor2TargetDistanceM :=
    MAX(0.0, machineConfig.sheetConveyor2LengthM);

sheetConveyor3TargetDistanceM :=
    MAX(0.0, machineConfig.sheetConveyor3LengthM);

sheetConveyor4TargetDistanceM :=
    MAX(0.0, machineConfig.sheetConveyor4LengthM);


//==============================================================
// 9) Check separation ready conditions
//==============================================================
// EN: Compare gap speed against base speed, not normal speed.
//     Otherwise operator speed-up would be incorrectly counted as gap opening.
packageGapReady :=
    speedControlEnabled AND
    (sheetConveyor2TargetDistanceM > 0.0) AND
    (sheetConveyor3TargetDistanceM > 0.0) AND
    (sheetConveyor4TargetDistanceM > 0.0) AND
    ((sheetConveyor2GapSpeedMPM - sheetConveyor2BaseSpeedMPM) >= machineConfig.minimumOpeningSpeedMPM) AND
    ((sheetConveyor3GapSpeedMPM - sheetConveyor3BaseSpeedMPM) >= machineConfig.minimumOpeningSpeedMPM) AND
    ((sheetConveyor4GapSpeedMPM - sheetConveyor4BaseSpeedMPM) >= machineConfig.minimumOpeningSpeedMPM);

sheetStackSeparationReady := packageGapReady;


//==============================================================
// 10) Sheet stack separation state machine
//==============================================================
IF NOT speedControlEnabled THEN

    sheetStackSeparationState      := 'DISABLED';
    sheetStackSeparationStateCode  := -1;

    packageSeparationState         := 0;

    sheetStackSeparationActive     := FALSE;
    sheetStackBrakeActive          := FALSE;
    brakeValve                     := FALSE;

    sheetConveyor2SeparationActive := FALSE;
    sheetConveyor3SeparationActive := FALSE;
    sheetConveyor4SeparationActive := FALSE;

    sheetConveyor2HighSpeedActive  := FALSE;
    sheetConveyor3HighSpeedActive  := FALSE;
    sheetConveyor4HighSpeedActive  := FALSE;

    sheetConveyor2OpeningDistanceM := 0.0;
    sheetConveyor3OpeningDistanceM := 0.0;
    sheetConveyor4OpeningDistanceM := 0.0;

    sheetConveyor1TargetSpeedMPM   := 0.0;
    sheetConveyor2TargetSpeedMPM   := 0.0;
    sheetConveyor3TargetSpeedMPM   := 0.0;
    sheetConveyor4TargetSpeedMPM   := 0.0;


ELSE

    CASE packageSeparationState OF

        0: // NORMAL
            sheetStackSeparationState     := 'NORMAL';
            sheetStackSeparationStateCode := 0;

            sheetStackSeparationActive    := FALSE;
            sheetStackBrakeActive         := FALSE;
            brakeValve                    := FALSE;

            sheetConveyor2SeparationActive := FALSE;
            sheetConveyor3SeparationActive := FALSE;
            sheetConveyor4SeparationActive := FALSE;

            sheetConveyor2HighSpeedActive  := FALSE;
            sheetConveyor3HighSpeedActive  := FALSE;
            sheetConveyor4HighSpeedActive  := FALSE;

            sheetConveyor2OpeningDistanceM := 0.0;
            sheetConveyor3OpeningDistanceM := 0.0;
            sheetConveyor4OpeningDistanceM := 0.0;

            sheetConveyor1TargetSpeedMPM  := sheetConveyor1BaseSpeedMPM;
            sheetConveyor2TargetSpeedMPM  := sheetConveyor2BaseSpeedMPM;
            sheetConveyor3TargetSpeedMPM  := sheetConveyor3BaseSpeedMPM;
            sheetConveyor4TargetSpeedMPM  := sheetConveyor4BaseSpeedMPM;

            // EN: Readiness is validated before the unload request is accepted.
            // PT: A prontidão é validada antes de o pedido de descarga ser aceito.
            IF dischargeRequestAccepted THEN
                packageSeparationState := 10;
            END_IF


        10: // START_SHEET_STACK_SEPARATION
            sheetStackSeparationState     := 'START_SEPARATION';
            sheetStackSeparationStateCode := 10;

            sheetStackSeparationActive    := TRUE;
            sheetStackSeparationStarted   := TRUE;

            sheetStackBrakeActive         := NOT changeBatchCycleActive;
            brakeValve                    := NOT changeBatchCycleActive;

            // EN: Conveyor 2 tracking starts immediately.
            sheetConveyor2SeparationStarted := TRUE;

            sheetConveyor2SeparationActive  := TRUE;
            sheetConveyor3SeparationActive  := FALSE;
            sheetConveyor4SeparationActive  := FALSE;

            // EN: Conveyor 2 and 3 accelerate together from the beginning.
            sheetConveyor2HighSpeedActive   := TRUE;
            sheetConveyor3HighSpeedActive   := TRUE;
            sheetConveyor4HighSpeedActive   := TRUE;

            sheetConveyor2OpeningDistanceM  := 0.0;
            sheetConveyor3OpeningDistanceM  := 0.0;
            sheetConveyor4OpeningDistanceM  := 0.0;

            IF changeBatchCycleActive THEN
                sheetConveyor1TargetSpeedMPM := sheetConveyor1GapSpeedMPM;
            ELSE
                sheetConveyor1TargetSpeedMPM := sheetConveyor1BaseSpeedMPM;
            END_IF;
            sheetConveyor2TargetSpeedMPM    := sheetConveyor2GapSpeedMPM;
            sheetConveyor3TargetSpeedMPM    := sheetConveyor3GapSpeedMPM;
            sheetConveyor4TargetSpeedMPM    := sheetConveyor4GapSpeedMPM;

            packageSeparationState := 20;


        20: // SHEET_CONVEYOR_2_SEPARATION_TRACKING
            sheetStackSeparationState     := 'CONV2_TRACKING';
            sheetStackSeparationStateCode := 20;

            sheetStackSeparationActive    := TRUE;

            sheetStackBrakeActive         := NOT changeBatchCycleActive;
            brakeValve                    := NOT changeBatchCycleActive;

            sheetConveyor2SeparationActive := TRUE;
            sheetConveyor3SeparationActive := FALSE;
            sheetConveyor4SeparationActive := FALSE;

            sheetConveyor2HighSpeedActive  := TRUE;
            sheetConveyor3HighSpeedActive  := TRUE;
            sheetConveyor4HighSpeedActive  := TRUE;

            IF changeBatchCycleActive THEN
                sheetConveyor1TargetSpeedMPM := sheetConveyor1GapSpeedMPM;
            ELSE
                sheetConveyor1TargetSpeedMPM := sheetConveyor1BaseSpeedMPM;
            END_IF;
            sheetConveyor2TargetSpeedMPM  := sheetConveyor2GapSpeedMPM;
            sheetConveyor3TargetSpeedMPM  := sheetConveyor3GapSpeedMPM;
            sheetConveyor4TargetSpeedMPM  := sheetConveyor4GapSpeedMPM;

            IF sheetConveyor2OpeningDistanceM >= sheetConveyor2TargetDistanceM THEN

                // EN: Conveyor 2 tracking finished. Conveyor 2 returns to base speed.
                sheetConveyor2SeparationFinished := TRUE;

                sheetConveyor2SeparationActive   := FALSE;
                sheetConveyor2HighSpeedActive    := FALSE;

                sheetStackBrakeActive            := FALSE;
                brakeValve                       := FALSE;

                sheetConveyor2TargetSpeedMPM     := sheetConveyor2BaseSpeedMPM;

                // EN: Conveyor 3 tracking starts after conveyor 2 returns to sync.
                sheetConveyor3SeparationStarted := TRUE;
                sheetConveyor3OpeningDistanceM  := 0.0;

                packageSeparationState := 30;

            END_IF


        30: // SHEET_CONVEYOR_3_SEPARATION_TRACKING
            sheetStackSeparationState     := 'CONV3_TRACKING';
            sheetStackSeparationStateCode := 30;

            sheetStackSeparationActive    := TRUE;

            sheetStackBrakeActive         := FALSE;
            brakeValve                    := FALSE;

            sheetConveyor2SeparationActive := FALSE;
            sheetConveyor3SeparationActive := TRUE;
            sheetConveyor4SeparationActive := FALSE;

            sheetConveyor2HighSpeedActive  := FALSE;
            sheetConveyor3HighSpeedActive  := TRUE;
            sheetConveyor4HighSpeedActive  := TRUE;

            sheetConveyor1TargetSpeedMPM  := sheetConveyor1BaseSpeedMPM;
            sheetConveyor2TargetSpeedMPM  := sheetConveyor2BaseSpeedMPM;
            sheetConveyor3TargetSpeedMPM  := sheetConveyor3GapSpeedMPM;
            sheetConveyor4TargetSpeedMPM  := sheetConveyor4GapSpeedMPM;

            IF sheetConveyor3OpeningDistanceM >= sheetConveyor3TargetDistanceM THEN

                // EN: Conveyor 3 returns to base synchronized speed.
                sheetConveyor3TargetSpeedMPM := sheetConveyor3BaseSpeedMPM;

                // EN: Conveyor 4 tracking starts after conveyor 3 returns to sync.
                // PT: O rastreamento da esteira 4 inicia após a esteira 3 retornar ao sincronismo.
                sheetConveyor4SeparationStarted := TRUE;
                sheetConveyor4OpeningDistanceM := 0.0;

                packageSeparationState := 40;

            END_IF


        40: // SHEET_CONVEYOR_4_SEPARATION_TRACKING
            sheetStackSeparationState     := 'CONV4_TRACKING';
            sheetStackSeparationStateCode := 40;

            sheetStackSeparationActive    := TRUE;
            sheetStackBrakeActive         := FALSE;
            brakeValve                    := FALSE;

            sheetConveyor2SeparationActive := FALSE;
            sheetConveyor3SeparationActive := FALSE;
            sheetConveyor4SeparationActive := TRUE;

            sheetConveyor2HighSpeedActive := FALSE;
            sheetConveyor3HighSpeedActive := FALSE;
            sheetConveyor4HighSpeedActive := TRUE;

            sheetConveyor1TargetSpeedMPM := sheetConveyor1BaseSpeedMPM;
            sheetConveyor2TargetSpeedMPM := sheetConveyor2BaseSpeedMPM;
            sheetConveyor3TargetSpeedMPM := sheetConveyor3BaseSpeedMPM;
            sheetConveyor4TargetSpeedMPM := sheetConveyor4GapSpeedMPM;

            IF sheetConveyor4OpeningDistanceM >= sheetConveyor4TargetDistanceM THEN
                sheetConveyor4TargetSpeedMPM := sheetConveyor4BaseSpeedMPM;
                packageSeparationState := 50;
            END_IF


        50: // FINISH_SHEET_STACK_SEPARATION
            sheetStackSeparationState     := 'FINISH_SEPARATION';
            sheetStackSeparationStateCode := 50;

            sheetStackSeparationActive    := FALSE;
            sheetStackSeparationFinished  := TRUE;

            sheetStackBrakeActive         := FALSE;
            brakeValve                    := FALSE;

            sheetConveyor2SeparationActive  := FALSE;
            sheetConveyor3SeparationActive  := FALSE;
            sheetConveyor4SeparationActive  := FALSE;

            sheetConveyor2HighSpeedActive   := FALSE;
            sheetConveyor3HighSpeedActive   := FALSE;
            sheetConveyor4HighSpeedActive   := FALSE;

            sheetConveyor3SeparationFinished := TRUE;
            sheetConveyor4SeparationFinished := TRUE;

            sheetConveyor1TargetSpeedMPM  := sheetConveyor1BaseSpeedMPM;
            sheetConveyor2TargetSpeedMPM  := sheetConveyor2BaseSpeedMPM;
            sheetConveyor3TargetSpeedMPM  := sheetConveyor3BaseSpeedMPM;
            sheetConveyor4TargetSpeedMPM  := sheetConveyor4BaseSpeedMPM;

            packageSeparationState := 0;


    ELSE

        packageSeparationState := 0;

    END_CASE;

END_IF;


//==============================================================
// 11) Limit speed targets
//==============================================================
sheetConveyor1TargetSpeedMPM := LIMIT(
    machineConfig.minimumSpeedMPM,
    sheetConveyor1TargetSpeedMPM,
    machineConfig.maximumSpeedMPM
);

sheetConveyor2TargetSpeedMPM := LIMIT(
    machineConfig.minimumSpeedMPM,
    sheetConveyor2TargetSpeedMPM,
    machineConfig.maximumSpeedMPM
);

sheetConveyor3TargetSpeedMPM := LIMIT(
    machineConfig.minimumSpeedMPM,
    sheetConveyor3TargetSpeedMPM,
    machineConfig.maximumSpeedMPM
);

sheetConveyor4TargetSpeedMPM := LIMIT(
    machineConfig.minimumSpeedMPM,
    sheetConveyor4TargetSpeedMPM,
    machineConfig.maximumSpeedMPM
);


//==============================================================
// 12) Ramp sheet conveyor 1 speed reference
//==============================================================
instRampSheetConveyor1(
    X          := sheetConveyor1TargetSpeedMPM,
    A_UP       := MAX(0.0, machineConfig.rampAccelerationUpMPMps2),
    A_DN       := -MAX(0.0, machineConfig.rampAccelerationDownMPMps2),
    VU_MAX     := MAX(0.0, machineConfig.rampVelocityUpMaxMPMps),
    VD_MAX     := -MAX(0.0, machineConfig.rampVelocityDownMaxMPMps),
    LIMIT_HIGH := machineConfig.maximumSpeedMPM,
    LIMIT_LOW  := machineConfig.minimumSpeedMPM,
    RST        := rampReset,
    Y          => sheetConveyor1SpeedRefMPM
);


//==============================================================
// 13) Ramp sheet conveyor 2 speed reference
//==============================================================
instRampSheetConveyor2(
    X          := sheetConveyor2TargetSpeedMPM,
    A_UP       := MAX(0.0, machineConfig.rampAccelerationUpMPMps2),
    A_DN       := -MAX(0.0, machineConfig.rampAccelerationDownMPMps2),
    VU_MAX     := MAX(0.0, machineConfig.rampVelocityUpMaxMPMps),
    VD_MAX     := -MAX(0.0, machineConfig.rampVelocityDownMaxMPMps),
    LIMIT_HIGH := machineConfig.maximumSpeedMPM,
    LIMIT_LOW  := machineConfig.minimumSpeedMPM,
    RST        := rampReset,
    Y          => sheetConveyor2SpeedRefMPM
);


//==============================================================
// 14) Ramp sheet conveyor 3 speed reference
//==============================================================
instRampSheetConveyor3(
    X          := sheetConveyor3TargetSpeedMPM,
    A_UP       := MAX(0.0, machineConfig.rampAccelerationUpMPMps2),
    A_DN       := -MAX(0.0, machineConfig.rampAccelerationDownMPMps2),
    VU_MAX     := MAX(0.0, machineConfig.rampVelocityUpMaxMPMps),
    VD_MAX     := -MAX(0.0, machineConfig.rampVelocityDownMaxMPMps),
    LIMIT_HIGH := machineConfig.maximumSpeedMPM,
    LIMIT_LOW  := machineConfig.minimumSpeedMPM,
    RST        := rampReset,
    Y          => sheetConveyor3SpeedRefMPM
);


//==============================================================
// 15) Ramp sheet conveyor 4 speed reference
//==============================================================
instRampSheetConveyor4(
    X          := sheetConveyor4TargetSpeedMPM,
    A_UP       := MAX(0.0, machineConfig.rampAccelerationUpMPMps2),
    A_DN       := -MAX(0.0, machineConfig.rampAccelerationDownMPMps2),
    VU_MAX     := MAX(0.0, machineConfig.rampVelocityUpMaxMPMps),
    VD_MAX     := -MAX(0.0, machineConfig.rampVelocityDownMaxMPMps),
    LIMIT_HIGH := machineConfig.maximumSpeedMPM,
    LIMIT_LOW  := machineConfig.minimumSpeedMPM,
    RST        := rampReset,
    Y          => sheetConveyor4SpeedRefMPM
);


//==============================================================
// 16) Calculate real separation tracking speed using ramped references
//==============================================================
// EN: Only the real speed differential above the base speed moves the
//     separation point through the conveyors.
//     Operator speed-up is already included in base speed, so it is not
//     counted as gap opening.
sheetConveyor2OpeningSpeedMPM :=
    MAX(0.0, sheetConveyor2SpeedRefMPM - sheetConveyor2BaseSpeedMPM);

sheetConveyor3OpeningSpeedMPM :=
    MAX(0.0, sheetConveyor3SpeedRefMPM - sheetConveyor3BaseSpeedMPM);

sheetConveyor4OpeningSpeedMPM :=
    MAX(0.0, sheetConveyor4SpeedRefMPM - sheetConveyor4BaseSpeedMPM);


//==============================================================
// 17) Integrate real separation tracking distance
//==============================================================
IF speedControlEnabled THEN

    IF packageSeparationState = 20 THEN

        IF sheetConveyor2OpeningSpeedMPM >= machineConfig.minimumOpeningSpeedMPM THEN

            sheetConveyor2OpeningDistanceM :=
                sheetConveyor2OpeningDistanceM +
                (sheetConveyor2OpeningSpeedMPM / 60.0) * scanTimeS;

        END_IF

    ELSIF packageSeparationState = 30 THEN

        IF sheetConveyor3OpeningSpeedMPM >= machineConfig.minimumOpeningSpeedMPM THEN

            sheetConveyor3OpeningDistanceM :=
                sheetConveyor3OpeningDistanceM +
                (sheetConveyor3OpeningSpeedMPM / 60.0) * scanTimeS;

        END_IF

    ELSIF packageSeparationState = 40 THEN

        IF sheetConveyor4OpeningSpeedMPM >= machineConfig.minimumOpeningSpeedMPM THEN

            sheetConveyor4OpeningDistanceM :=
                sheetConveyor4OpeningDistanceM +
                (sheetConveyor4OpeningSpeedMPM / 60.0) * scanTimeS;

        END_IF

    END_IF

END_IF;


//==============================================================
// 18) Publish tracking distances to outputs
//==============================================================
sheetConveyor2TrackingDistanceM := sheetConveyor2OpeningDistanceM;
sheetConveyor3TrackingDistanceM := sheetConveyor3OpeningDistanceM;
sheetConveyor4TrackingDistanceM := sheetConveyor4OpeningDistanceM;
END_METHOD

//==============================================================
// COMPLEX STACKER - ELEVATOR CONTROL
// EN: Controls homing, manual movement, automatic leveling,
//     discharge positioning and magnetic brake timing.
// PT: Controla homing, movimento manual, nivelamento automático,
//     posicionamento de descarga e temporização do freio magnético.
//
// Signed speed: positive = up; negative = down.
// Velocidade com sinal: positivo = subir; negativo = descer.
//
// State code:
// 0  = STOP
// 10 = HOME_DOWN_SEARCH
// 11 = HOME_RELEASE_SENSOR
// 12 = HOME_SETTLE
// 13 = HOME_SET_ENCODER
// 14 = HOME_WAIT_CLEAR_AND_MOVE_TO_UPPER_POSITION
// 20 = MANUAL
// 30 = AUTO_LEVELING
// 40 = DISCHARGE_POSITIONING
// 90 = FAULT
//==============================================================
METHOD _ElevatorControl
//==============================================================
// 1) Default internal commands
//==============================================================
elevatorSignedSpeedRefMmps := 0.0;
elevatorSetEncoderPositionTrigger := FALSE;
elevatorManualLowSpeedZoneActive := FALSE;
elevatorHomeDischargeConveyorRunRequest := FALSE;


//==============================================================
// 2) Homing request and lower sensor edge detection
//==============================================================
elevatorHomeRequestCombined :=
    systemRunEnable AND
    (
        elevatorHomeCmd OR
        (
            elevatorAutoCmd AND
            elevatorAutoHomeRequest
        )
    );

// EN: The automatic pulse is accepted directly so a maintained manual home
//     command cannot hide the mandatory start-triggered request.
// PT: O pulso automático é aceito diretamente para que um comando manual de
//     home mantido não esconda o pedido obrigatório gerado pela partida.
rElevatorHome :=
    (
        elevatorHomeRequestCombined AND
        NOT elevatorHomeRequestCombinedOld
    ) OR
    (
        systemRunEnable AND
        elevatorAutoCmd AND
        elevatorAutoHomeRequest
    );

elevatorHomeRequestCombinedOld := elevatorHomeRequestCombined;

elevatorHomeLimitReached := elevatorLowerLimit;

elevatorHomeLimitFallingEdge :=
    elevatorHomeLimitOld AND
    NOT elevatorHomeLimitReached;

elevatorHomeLimitOld := elevatorHomeLimitReached;


//==============================================================
// 2.1) Manual command rearm
//==============================================================
// EN: Manual commands held during homing or active discharge positioning
//     must be released before a new manual movement can start.
//     Waiting for stack separation keeps leveling and manual control active.
// PT: Comandos manuais mantidos durante homing ou posicionamento ativo de
//     descarte devem ser liberados antes que um novo movimento manual inicie.
//     A espera pela separação mantém o nivelamento e o controle manual ativos.
IF NOT systemRunEnable OR
   NOT safetyCircuitOk OR
   NOT elevatorDriveOk OR
   elevatorFault OR
   (
        (elevatorControlState >= 10) AND
        (elevatorControlState <= 14)
   ) OR
   (elevatorControlState = 40) OR
   (elevatorControlState = 90) OR
   elevatorTargetOverrideActive OR
   sheetStackDischargeActive THEN

    elevatorManualCommandArmed := FALSE;

ELSIF NOT elevatorUpCmd AND
      NOT elevatorDownCmd THEN

    elevatorManualCommandArmed := TRUE;

END_IF;

elevatorManualCommandRequest :=
    elevatorManualCommandArmed AND
    (elevatorUpCmd OR elevatorDownCmd);


//==============================================================
// 3) Movement permissions
//==============================================================
elevatorUpAllowed :=
    systemRunEnable AND
    safetyCircuitOk AND
    elevatorDriveOk AND
    NOT elevatorUpperLimit AND
    NOT elevatorUpperSafetyLimit AND
    NOT backstopMaterialInterlockSensor AND
    (
        (NOT elevatorHomed) OR
        (elevatorPositionMm < machineConfig.elevatorMaxPositionMm)
    );

elevatorDownAllowed :=
    systemRunEnable AND
    safetyCircuitOk AND
    elevatorDriveOk AND
    NOT elevatorLowerLimit AND
    NOT elevatorLowerSafetyLimit AND
    (
        (NOT elevatorHomed) OR
        (elevatorPositionMm > machineConfig.elevatorMinPositionMm)
    );

// EN: Homing search ignores the normal lower limit until it is detected.
// PT: A busca de home ignora o limite inferior normal até detectá-lo.
elevatorHomeDownAllowed :=
    systemRunEnable AND
    safetyCircuitOk AND
    elevatorDriveOk AND
    NOT elevatorLowerSafetyLimit;

// EN: Upward release respects the backstop material interlock.
// PT: A liberação para cima respeita o intertravamento de material do backstop.
elevatorHomeReleaseAllowed :=
    systemRunEnable AND
    safetyCircuitOk AND
    elevatorDriveOk AND
    NOT elevatorUpperLimit AND
    NOT elevatorUpperSafetyLimit AND
    NOT backstopMaterialInterlockSensor;

//==============================================================
// 4) Target and position feedback
//==============================================================
IF elevatorControlState = 14 THEN

    elevatorTargetPositionMm := machineConfig.elevatorMaxPositionMm;

ELSIF elevatorTargetOverrideActive THEN

    elevatorTargetPositionMm :=
        LIMIT(
            machineConfig.elevatorMinPositionMm,
            elevatorTargetOverridePositionMm,
            machineConfig.elevatorMaxPositionMm
        );

ELSE

    elevatorTargetPositionMm :=
        LIMIT(
            machineConfig.elevatorMinPositionMm,
            elevatorPositionMm,
            machineConfig.elevatorMaxPositionMm
        );

END_IF;

elevatorPositionErrorMm :=
    elevatorTargetPositionMm - elevatorPositionMm;

elevatorAbsPositionErrorMm := ABS(elevatorPositionErrorMm);

// EN: Proportional position control with independent directional limits.
//     No minimum speed is forced; the servo may receive zero near the target.
// PT: Controle proporcional de posição com limites independentes por sentido.
//     Não força velocidade mínima; o servo pode receber zero próximo ao alvo.
elevatorRawSpeedRefMmps :=
    elevatorPositionErrorMm * MAX(0.0, machineConfig.elevatorPositionKp);

elevatorRawSpeedRefMmps :=
    LIMIT(
        -ABS(machineConfig.elevatorAutomaticDownSpeedMmps),
        elevatorRawSpeedRefMmps,
        ABS(machineConfig.elevatorAutomaticUpSpeedMmps)
    );

// EN: Endpoint flags depend on actual feedback and remain valid
//     independently of the active automatic target.
// PT: As flags de extremidade dependem do feedback real e permanecem
//     válidas independentemente do alvo automático ativo.
elevatorAtMinPosition :=
    elevatorHomed AND
    (
        elevatorLowerLimit OR
        (
            elevatorPositionMm <=
            (
                machineConfig.elevatorMinPositionMm +
                MAX(0.0, machineConfig.elevatorPositionToleranceMm)
            )
        )
    );

elevatorAtMaxPosition :=
    elevatorHomed AND
    (
        elevatorUpperLimit OR
        (
            elevatorPositionMm >=
            (
                machineConfig.elevatorMaxPositionMm -
                MAX(0.0, machineConfig.elevatorPositionToleranceMm)
            )
        )
    );

elevatorInPosition :=
    elevatorHomed AND
    (
        (elevatorAbsPositionErrorMm <= machineConfig.elevatorPositionToleranceMm)
        OR
        (
            elevatorUpperLimit AND
            (elevatorTargetPositionMm >= machineConfig.elevatorMaxPositionMm)
        )
        OR
        (
            elevatorLowerLimit AND
            (elevatorTargetPositionMm <= machineConfig.elevatorMinPositionMm)
        )
    );


//==============================================================
// 5) Fault reset
//==============================================================
IF resetCmd AND
   safetyCircuitOk AND
   elevatorDriveOk AND
   NOT elevatorUpperSafetyLimit AND
   NOT elevatorLowerSafetyLimit THEN

    elevatorFault := FALSE;
    elevatorFaultCode := 0;

    IF elevatorControlState = 90 THEN
        elevatorControlState := 0;
    END_IF

END_IF;


//==============================================================
// 6) Invalidate an interrupted homing sequence
//==============================================================
// EN: If homing or its final upward movement is interrupted by a
//     protection/system stop, a new homing cycle is required.
// PT: Se o homing ou sua subida final for interrompido por proteção/parada,
//     um novo ciclo de homing será obrigatório.
IF (elevatorControlState >= 10) AND
   (elevatorControlState <= 14) AND
   (
       NOT systemRunEnable OR
       NOT safetyCircuitOk OR
       NOT elevatorDriveOk OR
       elevatorUpperSafetyLimit OR
       elevatorLowerSafetyLimit
   ) THEN

    elevatorHomed := FALSE;
    elevatorReadyForAutomaticCycle := FALSE;

END_IF;


//==============================================================
// 7) General protection
//==============================================================
IF NOT safetyCircuitOk THEN

    elevatorState := 'SAFETY_OFF';
    elevatorFault := TRUE;
    elevatorFaultCode := 2;
    elevatorControlState := 90;

    tonElevatorHomingTimeout(IN := FALSE);
    tonElevatorHomeSettleDelay(IN := FALSE);
    tonElevatorLevelingSpeed2Delay(IN := FALSE);


ELSIF NOT elevatorDriveOk THEN

    elevatorState := 'DRIVE_NOT_OK';
    elevatorFault := TRUE;
    elevatorFaultCode := 1;
    elevatorControlState := 90;

    tonElevatorHomingTimeout(IN := FALSE);
    tonElevatorHomeSettleDelay(IN := FALSE);
    tonElevatorLevelingSpeed2Delay(IN := FALSE);


ELSIF elevatorUpperSafetyLimit THEN

    elevatorState := 'UPPER_SAFE_LIMIT';
    elevatorFault := TRUE;
    elevatorFaultCode := 4;
    elevatorControlState := 90;

    tonElevatorHomingTimeout(IN := FALSE);
    tonElevatorHomeSettleDelay(IN := FALSE);
    tonElevatorLevelingSpeed2Delay(IN := FALSE);


ELSIF elevatorLowerSafetyLimit THEN

    elevatorState := 'LOWER_SAFE_LIMIT';
    elevatorFault := TRUE;
    elevatorFaultCode := 5;
    elevatorControlState := 90;

    tonElevatorHomingTimeout(IN := FALSE);
    tonElevatorHomeSettleDelay(IN := FALSE);
    tonElevatorLevelingSpeed2Delay(IN := FALSE);


ELSIF NOT systemRunEnable THEN

    elevatorState := 'SYSTEM_DISABLED';
    elevatorSignedSpeedRefMmps := 0.0;

    tonElevatorHomingTimeout(IN := FALSE);
    tonElevatorHomeSettleDelay(IN := FALSE);
    tonElevatorLevelingSpeed2Delay(IN := FALSE);

    IF elevatorControlState <> 90 THEN
        elevatorControlState := 0;
    END_IF


ELSE

    //==========================================================
    // 8) Mode selection
    //==========================================================
    // EN: A new home command is ignored while discharge is active/pending.
    // PT: Novo comando de home é ignorado durante descarte ativo/pendente.
    IF rElevatorHome AND
       NOT elevatorFault AND
       NOT sheetStackDischargeActive AND
       NOT sheetStackDischargePending THEN

        elevatorControlState := 10;

        // EN: Consume the pending request only after homing is accepted.
        // PT: Consome o pedido pendente somente após o homing ser aceito.
        elevatorAutoHomePending := FALSE;

    END_IF;

    // EN: Discharge override blocks manual and leveling commands.
    // PT: Override de descarte bloqueia comandos manuais e nivelamento.
    IF elevatorTargetOverrideActive AND
       elevatorHomed AND
       (elevatorControlState <> 10) AND
       (elevatorControlState <> 11) AND
       (elevatorControlState <> 12) AND
       (elevatorControlState <> 13) AND
       (elevatorControlState <> 14) AND
       (elevatorControlState <> 90) THEN

        elevatorControlState := 40;

    END_IF;


    //==========================================================
    // 9) Elevator state machine
    //==========================================================
    CASE elevatorControlState OF

        0: // STOP
            elevatorState := 'STOP';

            tonElevatorHomingTimeout(IN := FALSE);
            tonElevatorHomeSettleDelay(IN := FALSE);
            tonElevatorLevelingSpeed2Delay(IN := FALSE);

            // EN: Manual movement is available with automatic mode off.
            //     With automatic mode on, it is available only after homing
            //     and completion of the upper home positioning.
            // PT: O movimento manual fica disponível com o automático desligado.
            //     Com o automático ligado, fica disponível somente após o homing
            //     e a conclusão do posicionamento superior.
            IF elevatorManualCommandRequest AND
               (
                   NOT elevatorAutoCmd OR
                   (
                       elevatorHomed AND
                       elevatorReadyForAutomaticCycle
                   )
               ) THEN

                elevatorControlState := 20;

            ELSIF elevatorAutoCmd AND
                  elevatorHomed AND
                  elevatorReadyForAutomaticCycle THEN

                elevatorControlState := 30;

            END_IF


        10: // HOME_DOWN_SEARCH
            elevatorState := 'HOME_DOWN';
            elevatorHomed := FALSE;
            elevatorReadyForAutomaticCycle := FALSE;
            elevatorInPosition := FALSE;
            elevatorHomeDischargeComplete := FALSE;

            tonElevatorHomingTimeout(
                IN := TRUE,
                PT := machineConfig.elevatorHomingTimeout
            );

            IF tonElevatorHomingTimeout.Q THEN

                elevatorSignedSpeedRefMmps := 0.0;
                tonElevatorHomingTimeout(IN := FALSE);

                elevatorFault := TRUE;
                elevatorFaultCode := 3;
                elevatorState := 'HOME_TIMEOUT';
                elevatorControlState := 90;

            ELSIF elevatorHomeLimitReached THEN

                elevatorSignedSpeedRefMmps := 0.0;
                tonElevatorHomingTimeout(IN := FALSE);

                // EN: Start clearing the platform as soon as the lower home
                //     limit is reached. Homing continues through encoder reset.
                // PT: Inicia a limpeza da plataforma assim que o limite inferior
                //     do home é atingido. O homing continua até zerar o encoder.
                elevatorHomeDischargeConveyorRunRequest := TRUE;
                elevatorControlState := 11;

            ELSIF elevatorHomeDownAllowed THEN

                elevatorSignedSpeedRefMmps :=
                    -ABS(machineConfig.elevatorHomingSpeedMmps);

            END_IF


        11: // HOME_RELEASE_SENSOR
            elevatorState := 'HOME_RELEASE';
            elevatorHomeDischargeConveyorRunRequest := TRUE;

            tonElevatorHomingTimeout(
                IN := TRUE,
                PT := machineConfig.elevatorHomingTimeout
            );

            IF tonElevatorHomingTimeout.Q THEN

                elevatorSignedSpeedRefMmps := 0.0;
                tonElevatorHomingTimeout(IN := FALSE);

                elevatorFault := TRUE;
                elevatorFaultCode := 3;
                elevatorState := 'HOME_TIMEOUT';
                elevatorControlState := 90;

            ELSIF elevatorHomeLimitFallingEdge THEN

                elevatorSignedSpeedRefMmps := 0.0;
                tonElevatorHomingTimeout(IN := FALSE);
                tonElevatorHomeSettleDelay(IN := FALSE);
                elevatorControlState := 12;

            ELSIF elevatorHomeReleaseAllowed THEN

                elevatorSignedSpeedRefMmps :=
                    ABS(machineConfig.elevatorHomingReleaseSpeedMmps);

            END_IF


        12: // HOME_SETTLE
            elevatorState := 'HOME_SETTLE';
            elevatorSignedSpeedRefMmps := 0.0;
            elevatorHomeDischargeConveyorRunRequest := TRUE;

            // EN: Encoder reset is allowed only while the lower sensor
            //     remains released throughout the settle time.
            // PT: Reset do encoder é permitido somente se o sensor inferior
            //     permanecer livre durante todo o tempo de estabilização.
            IF elevatorHomeLimitReached THEN

                tonElevatorHomeSettleDelay(IN := FALSE);
                elevatorControlState := 11;

            ELSE

                tonElevatorHomeSettleDelay(
                    IN := TRUE,
                    PT := machineConfig.elevatorHomeSettleDelay
                );

                IF tonElevatorHomeSettleDelay.Q THEN
                    tonElevatorHomeSettleDelay(IN := FALSE);
                    elevatorControlState := 13;
                END_IF

            END_IF


        13: // HOME_SET_ENCODER
            elevatorState := 'HOME_SET_ENCODER';
            elevatorSignedSpeedRefMmps := 0.0;
            elevatorHomeDischargeConveyorRunRequest := TRUE;

            elevatorSetEncoderPositionTrigger := TRUE;
            elevatorSetEncoderPositionMm := machineConfig.elevatorHomePositionMm;

            elevatorHomed := TRUE;
            elevatorFault := FALSE;
            elevatorFaultCode := 0;

            tonElevatorHomingTimeout(IN := FALSE);
            elevatorControlState := 14;


        14: // HOME_MOVE_TO_UPPER_POSITION
            tonElevatorHomingTimeout(
                IN := TRUE,
                PT := machineConfig.elevatorHomingTimeout
            );

            // EN: Keep the conveyor running after the encoder is set. The final
            //     upward movement is released only after the actual run time and
            //     both platform-clear conditions are confirmed.
            // PT: Mantém a esteira ligada após zerar o encoder. A subida final é
            //     liberada somente após confirmar o tempo real de giro e as duas
            //     condições de plataforma livre.
            IF NOT elevatorHomeDischargeComplete THEN

                elevatorState := 'HOME_WAIT_CLEAR';
                elevatorHomeDischargeConveyorRunRequest := TRUE;

                IF tonElevatorHomeDischargeMinimumRun.Q AND
                   elevatorStackExitClearSensor AND
						elevatorStackPresentSensor THEN

                    elevatorHomeDischargeComplete := TRUE;
                    elevatorHomeDischargeConveyorRunRequest := FALSE;
                    elevatorState := 'HOME_MOVE_UP';

                END_IF

            ELSE

                elevatorState := 'HOME_MOVE_UP';

            END_IF;


            IF elevatorInPosition AND
               elevatorHomeDischargeComplete THEN

                elevatorSignedSpeedRefMmps := 0.0;
                tonElevatorHomingTimeout(IN := FALSE);
                elevatorReadyForAutomaticCycle := TRUE;

                IF elevatorAutoCmd THEN
                    elevatorControlState := 30;
                ELSE
                    elevatorControlState := 0;
                END_IF

            ELSIF tonElevatorHomingTimeout.Q THEN

                elevatorSignedSpeedRefMmps := 0.0;
                tonElevatorHomingTimeout(IN := FALSE);

                elevatorHomed := FALSE;
                elevatorReadyForAutomaticCycle := FALSE;
                elevatorFault := TRUE;
                elevatorFaultCode := 3;
                elevatorState := 'HOME_UP_TIMEOUT';
                elevatorControlState := 90;

            ELSIF elevatorHomeDischargeComplete AND
                  (elevatorRawSpeedRefMmps > 0.0) AND
                  elevatorUpAllowed THEN

                elevatorSignedSpeedRefMmps :=
                    elevatorRawSpeedRefMmps;

            ELSIF elevatorHomeDischargeComplete AND
                  (elevatorRawSpeedRefMmps < 0.0) AND
                  elevatorDownAllowed THEN

                elevatorSignedSpeedRefMmps :=
                    elevatorRawSpeedRefMmps;

            END_IF


        20: // MANUAL
            elevatorState := 'MANUAL';

            tonElevatorHomingTimeout(IN := FALSE);
            tonElevatorHomeSettleDelay(IN := FALSE);
            tonElevatorLevelingSpeed2Delay(IN := FALSE);

            // EN: Waiting for stack separation does not cancel manual operation.
            //     Active positioning or an elevator override cancels it.
            // PT: A espera pela separação da pilha não cancela a operação manual.
            //     O posicionamento ativo ou um override do elevador a cancela.
            IF sheetStackDischargeActive OR
               elevatorTargetOverrideActive THEN

                elevatorSignedSpeedRefMmps := 0.0;

                IF elevatorAutoCmd AND
                   elevatorHomed AND
                   elevatorReadyForAutomaticCycle THEN

                    elevatorControlState := 30;

                ELSE

                    elevatorControlState := 0;

                END_IF


            ELSIF elevatorAutoCmd AND
                  (
                      NOT elevatorHomed OR
                      NOT elevatorReadyForAutomaticCycle
                  ) THEN

                elevatorSignedSpeedRefMmps := 0.0;
                elevatorState := 'AUTO_NO_HOME';
                elevatorControlState := 0;

            ELSIF elevatorUpCmd AND elevatorDownCmd THEN

                elevatorSignedSpeedRefMmps := 0.0;

            ELSIF elevatorUpCmd THEN

                IF elevatorUpAllowed THEN

                    // EN: Reduce manual upward speed only while approaching
                    //     the configured maximum position.
                    // PT: Reduz a velocidade manual de subida somente durante
                    //     a aproximação da posição máxima configurada.
                    elevatorManualLowSpeedZoneActive :=
                        elevatorHomed AND
                        (
                            LIMIT(
                                0.0,
                                machineConfig.elevatorManualLowSpeedFactor,
                                1.0
                            ) < 1.0
                        ) AND
                        (
                            elevatorPositionMm >=
                            (
                                machineConfig.elevatorMaxPositionMm -
                                MAX(
                                    0.0,
                                    machineConfig.elevatorManualLowSpeedZoneMm
                                )
                            )
                        );

                    IF elevatorManualLowSpeedZoneActive THEN

                        elevatorSignedSpeedRefMmps :=
                            ABS(machineConfig.elevatorManualSpeedMmps) *
                            LIMIT(
                                0.0,
                                machineConfig.elevatorManualLowSpeedFactor,
                                1.0
                            );

                    ELSE

                        elevatorSignedSpeedRefMmps :=
                            ABS(machineConfig.elevatorManualSpeedMmps);

                    END_IF

                ELSE
                    elevatorSignedSpeedRefMmps := 0.0;
                END_IF

            ELSIF elevatorDownCmd THEN

                IF elevatorDownAllowed THEN

                    // EN: Reduce manual downward speed only while approaching
                    //     the configured minimum position.
                    // PT: Reduz a velocidade manual de descida somente durante
                    //     a aproximação da posição mínima configurada.
                    elevatorManualLowSpeedZoneActive :=
                        elevatorHomed AND
                        (
                            LIMIT(
                                0.0,
                                machineConfig.elevatorManualLowSpeedFactor,
                                1.0
                            ) < 1.0
                        ) AND
                        (
                            elevatorPositionMm <=
                            (
                                machineConfig.elevatorMinPositionMm +
                                MAX(
                                    0.0,
                                    machineConfig.elevatorManualLowSpeedZoneMm
                                )
                            )
                        );

                    IF elevatorManualLowSpeedZoneActive THEN

                        elevatorSignedSpeedRefMmps :=
                            -ABS(machineConfig.elevatorManualSpeedMmps) *
                            LIMIT(
                                0.0,
                                machineConfig.elevatorManualLowSpeedFactor,
                                1.0
                            );

                    ELSE

                        elevatorSignedSpeedRefMmps :=
                            -ABS(machineConfig.elevatorManualSpeedMmps);

                    END_IF

                ELSE
                    elevatorSignedSpeedRefMmps := 0.0;
                END_IF

            ELSE

                elevatorSignedSpeedRefMmps := 0.0;

                // EN: When manual intervention ends, automatic leveling
                //     may immediately evaluate the current level sensor.
                // PT: Ao terminar a intervenção manual, o nivelamento
                //     automático pode avaliar imediatamente o sensor atual.
                IF elevatorAutoCmd AND
                   elevatorHomed AND
                   elevatorReadyForAutomaticCycle THEN

                    elevatorControlState := 30;

                ELSE

                    elevatorControlState := 0;

                END_IF

            END_IF


        30: // AUTO_LEVELING
            elevatorState := 'AUTO_LEVELING';

            tonElevatorHomingTimeout(IN := FALSE);
            tonElevatorHomeSettleDelay(IN := FALSE);

            IF NOT elevatorAutoCmd THEN

                elevatorSignedSpeedRefMmps := 0.0;
                tonElevatorLevelingSpeed2Delay(IN := FALSE);
                elevatorControlState := 0;

            ELSIF NOT elevatorHomed OR
                  NOT elevatorReadyForAutomaticCycle THEN

                elevatorSignedSpeedRefMmps := 0.0;
                tonElevatorLevelingSpeed2Delay(IN := FALSE);
                elevatorState := 'AUTO_NO_HOME';

            ELSIF (elevatorUpCmd OR elevatorDownCmd) AND
                  NOT elevatorManualCommandArmed THEN

                // EN: A command held from homing or discharge inhibits
                //     leveling but cannot start a manual movement.
                // PT: Um comando mantido desde o homing ou descarte bloqueia
                //     o nivelamento, mas não pode iniciar movimento manual.
                elevatorSignedSpeedRefMmps := 0.0;
                tonElevatorLevelingSpeed2Delay(IN := FALSE);

            // EN: Manual correction remains available while the discharge
            //     sequence is waiting for stack separation.
            // PT: A correção manual permanece disponível enquanto a sequência
            //     de descarte aguarda a separação da pilha.
            ELSIF elevatorManualCommandRequest AND
                  NOT sheetStackDischargeActive AND
                  NOT elevatorTargetOverrideActive THEN

                // EN: Manual commands have priority over the level sensor.
                //     The speed-2 delay restarts after manual intervention.
                // PT: Os comandos manuais têm prioridade sobre o sensor de nível.
                //     O atraso da velocidade 2 reinicia após a intervenção manual.
                elevatorSignedSpeedRefMmps := 0.0;
                tonElevatorLevelingSpeed2Delay(IN := FALSE);
                elevatorControlState := 20;

            ELSIF backstopStackLevelSensor AND
                  elevatorDownAllowed THEN

                tonElevatorLevelingSpeed2Delay(
                    IN := TRUE,
                    PT := machineConfig.elevatorLevelingSpeed2Delay
                );

                IF tonElevatorLevelingSpeed2Delay.Q THEN
                    elevatorSignedSpeedRefMmps :=
                        -ABS(machineConfig.elevatorLevelingSpeed2Mmps);
                ELSE
                    elevatorSignedSpeedRefMmps :=
                        -ABS(machineConfig.elevatorLevelingSpeed1Mmps);
                END_IF

            ELSE

                elevatorSignedSpeedRefMmps := 0.0;
                tonElevatorLevelingSpeed2Delay(IN := FALSE);

            END_IF


        40: // DISCHARGE_POSITIONING
            elevatorState := 'DISCHARGE_POSITION';

            tonElevatorLevelingSpeed2Delay(IN := FALSE);

            IF NOT elevatorTargetOverrideActive THEN

                elevatorSignedSpeedRefMmps := 0.0;

                IF elevatorAutoCmd AND
                   elevatorHomed AND
                   elevatorReadyForAutomaticCycle THEN

                    elevatorControlState := 30;

                ELSE

                    elevatorControlState := 0;

                END_IF

            ELSIF elevatorInPosition THEN

                elevatorSignedSpeedRefMmps := 0.0;

            ELSIF (elevatorRawSpeedRefMmps > 0.0) AND elevatorUpAllowed THEN

                elevatorSignedSpeedRefMmps :=
                    elevatorRawSpeedRefMmps;

            ELSIF (elevatorRawSpeedRefMmps < 0.0) AND elevatorDownAllowed THEN

                elevatorSignedSpeedRefMmps :=
                    elevatorRawSpeedRefMmps;

            END_IF


        90: // FAULT
            elevatorState := 'FAULT';
            elevatorSignedSpeedRefMmps := 0.0;

            tonElevatorHomingTimeout(IN := FALSE);
            tonElevatorHomeSettleDelay(IN := FALSE);
            tonElevatorLevelingSpeed2Delay(IN := FALSE);


        ELSE
            elevatorControlState := 0;

    END_CASE;

END_IF;


// EN: Any transition outside the homing states cancels its conveyor request
//     in the same scan, including stop, fault and completed homing.
// PT: Qualquer transição para fora dos estados de homing cancela o pedido da
//     esteira no mesmo scan, incluindo parada, falha e homing concluído.
IF (elevatorControlState < 10) OR
   (elevatorControlState > 14) THEN

    elevatorHomeDischargeConveyorRunRequest := FALSE;
    elevatorHomeDischargeComplete := FALSE;

END_IF;


//==============================================================
// 10) Elevator home discharge conveyor minimum run time
//==============================================================
// EN: Count only while the homing request is active and the conveyor run output
//     was commanded TRUE. Reading the previous scan adds a conservative delay.
// PT: Conta somente enquanto o pedido do homing estiver ativo e a saída de giro
//     da esteira tiver sido comandada. A leitura do scan anterior adiciona atraso.
tonElevatorHomeDischargeMinimumRun(
    IN :=
        elevatorHomeDischargeConveyorRunRequest AND
        sheetStackDischargeConveyorRun,
    PT := machineConfig.sheetStackDischargeTime
);


//==============================================================
// 11) Encoder set pulse
//==============================================================
tpElevatorSetEncoderPosition(
    IN := elevatorSetEncoderPositionTrigger,
    PT := machineConfig.elevatorSetEncoderPulseTime
);

elevatorSetEncoderPosition := tpElevatorSetEncoderPosition.Q;


